// SIMATIC S7-200 SMART project (STEP 7-Micro/WIN SMART), CPU ST40

SYMBOL_TABLE Table 1
Move_X           Q0.0
Move_Z           Q0.1
Grab             Q0.2
Lids_conveyor    Q0.3
Clamp_lid        Q0.4
Pos_raise_lids   Q0.5
Bases_conveyor   Q0.6
Clamp_base       Q0.7
Pos_raise_bases  Q1.0
Strat_light      Q1.1
Reset_light      Q1.2
Stop_light       Q1.3
Counter          QW4
Moving_X         V0.0
Lid_at_place     V0.1
Item_detected    V0.2
Moving_Z         V0.3
Lid_clamped      V0.4
Pos_at_limit_lids V0.5
Base_at_place    V0.6
Base_clamped     V0.7
Pos_at_limit_bases V1.0
Part_leaving     V1.1
Start            V1.2
Reset            V1.3
Stop_            V1.4
Emergency_stop   V1.5
END_SYMBOL_TABLE

SYMBOL_TABLE System Symbols
Always_On        SM0.0    // Always ON
END_SYMBOL_TABLE

ORGANIZATION_BLOCK MAIN:OB1
TITLE=Program Comments
BEGIN
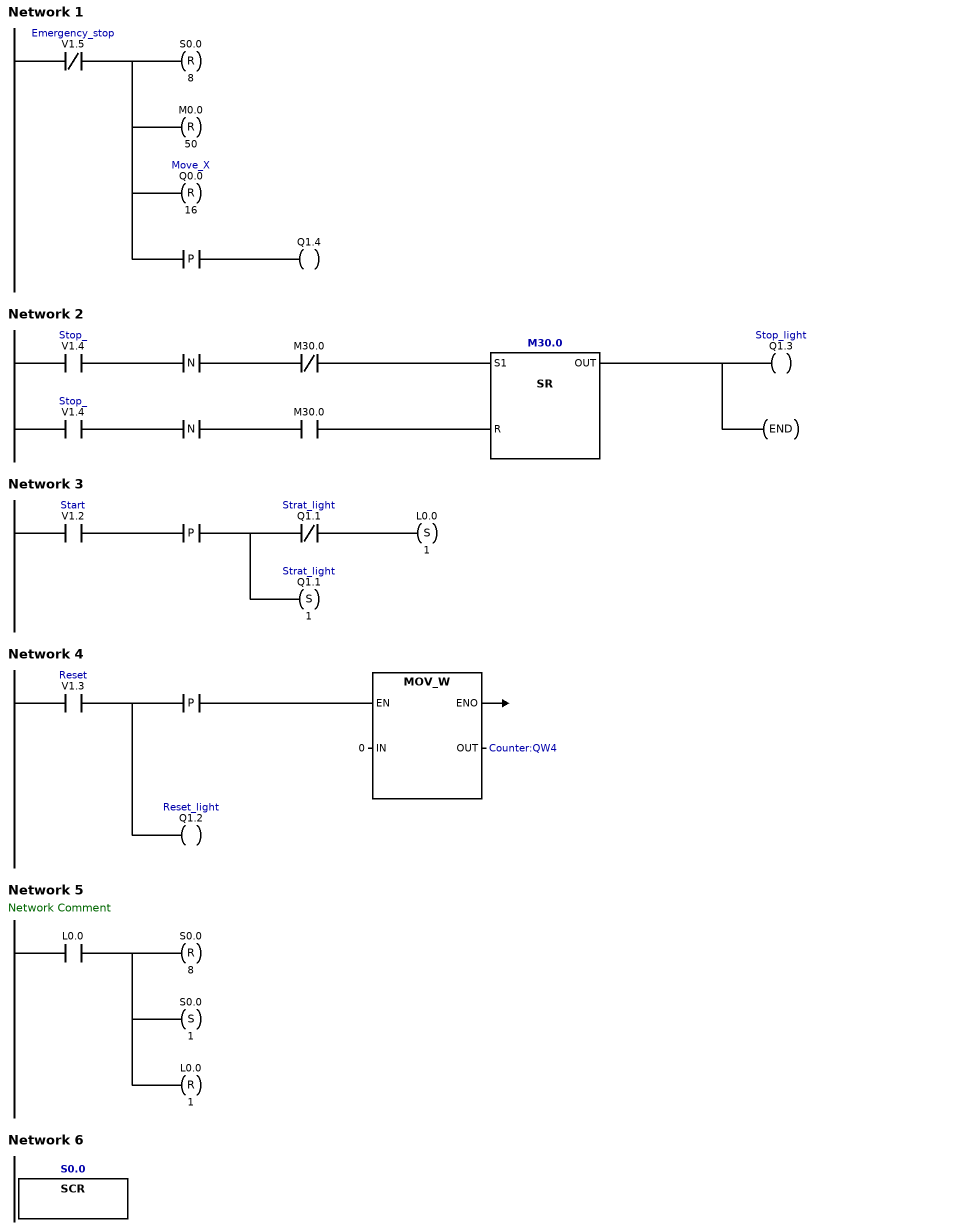
Network 1
LDN    Emergency_stop:V1.5
R      S0.0, 8
R      M0.0, 50
R      Move_X:Q0.0, 16
EU
=      Q1.4
Network 2
LD     Stop_:V1.4
ED
AN     M30.0
LD     Stop_:V1.4
ED
A      M30.0
NOT
A      M30.0
OLD
=      M30.0
=      Stop_light:Q1.3
END
Network 3
LD     Start:V1.2
EU
LPS
AN     Strat_light:Q1.1
S      L0.0, 1
LPP
S      Strat_light:Q1.1, 1
Network 4
LD     Reset:V1.3
LPS
EU
MOVW   0, Counter:QW4
LPP
=      Reset_light:Q1.2
Network 5
// Network Comment
LD     L0.0
R      S0.0, 8
S      S0.0, 1
R      L0.0, 1
Network 6
LSCR   S0.0
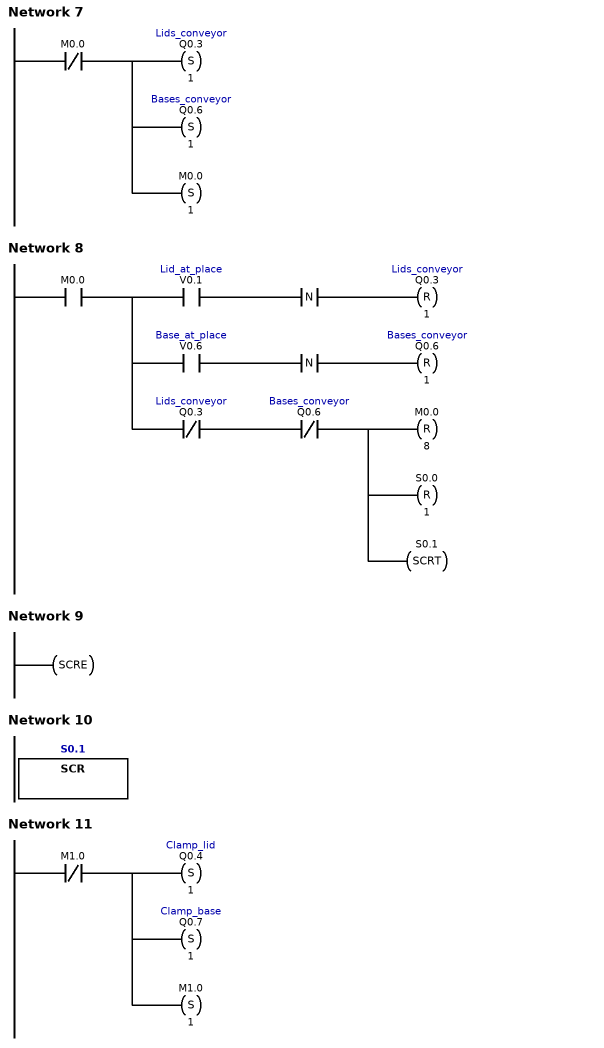
Network 7
LDN    M0.0
S      Lids_conveyor:Q0.3, 1
S      Bases_conveyor:Q0.6, 1
S      M0.0, 1
Network 8
LD     M0.0
LPS
A      Lid_at_place:V0.1
ED
R      Lids_conveyor:Q0.3, 1
LRD
A      Base_at_place:V0.6
ED
R      Bases_conveyor:Q0.6, 1
LPP
AN     Lids_conveyor:Q0.3
AN     Bases_conveyor:Q0.6
R      M0.0, 8
R      S0.0, 1
SCRT   S0.1
Network 9
SCRE
Network 10
LSCR   S0.1
Network 11
LDN    M1.0
S      Clamp_lid:Q0.4, 1
S      Clamp_base:Q0.7, 1
S      M1.0, 1
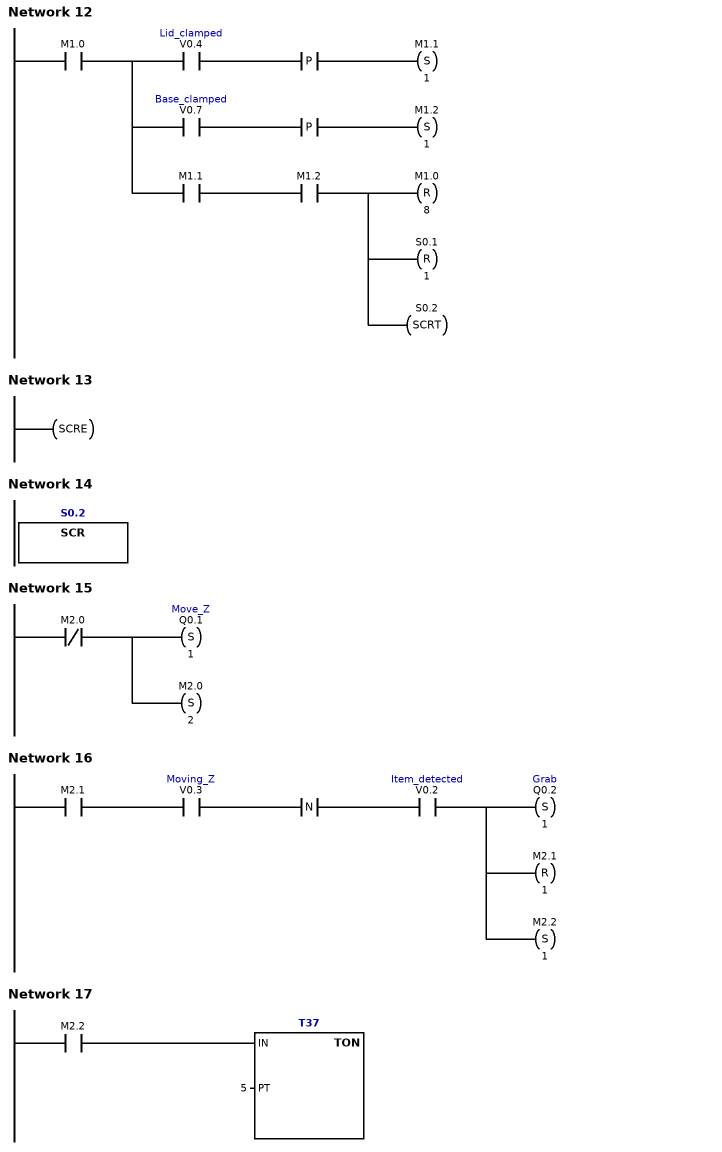
Network 12
LD     M1.0
LPS
A      Lid_clamped:V0.4
EU
S      M1.1, 1
LRD
A      Base_clamped:V0.7
EU
S      M1.2, 1
LPP
A      M1.1
A      M1.2
R      M1.0, 8
R      S0.1, 1
SCRT   S0.2
Network 13
SCRE
Network 14
LSCR   S0.2
Network 15
LDN    M2.0
S      Move_Z:Q0.1, 1
S      M2.0, 2
Network 16
LD     M2.1
A      Moving_Z:V0.3
ED
A      Item_detected:V0.2
S      Grab:Q0.2, 1
R      M2.1, 1
S      M2.2, 1
Network 17
LD     M2.2
TON    T37, 5
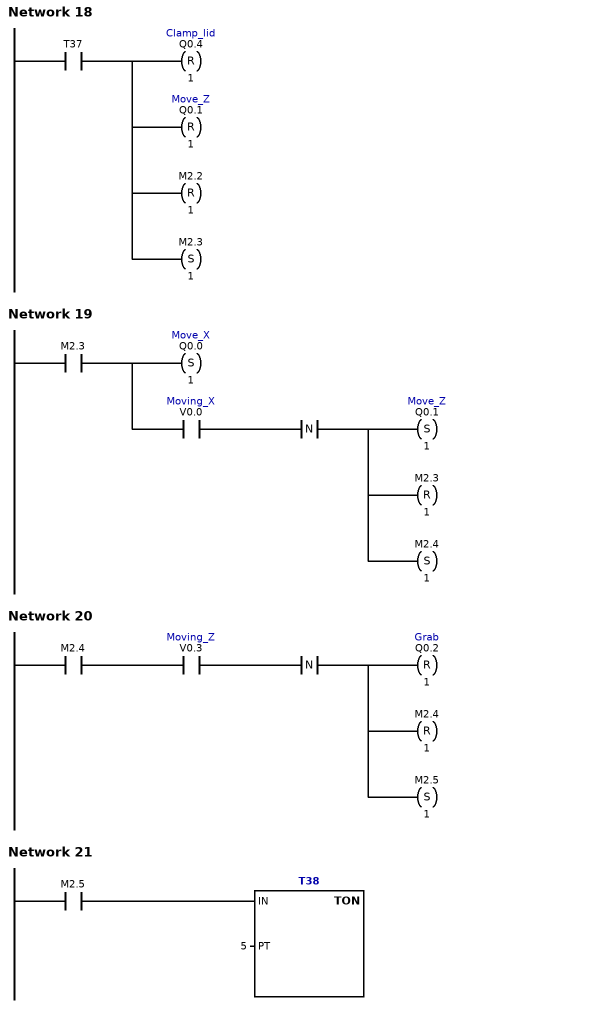
Network 18
LD     T37
R      Clamp_lid:Q0.4, 1
R      Move_Z:Q0.1, 1
R      M2.2, 1
S      M2.3, 1
Network 19
LD     M2.3
S      Move_X:Q0.0, 1
A      Moving_X:V0.0
ED
S      Move_Z:Q0.1, 1
R      M2.3, 1
S      M2.4, 1
Network 20
LD     M2.4
A      Moving_Z:V0.3
ED
R      Grab:Q0.2, 1
R      M2.4, 1
S      M2.5, 1
Network 21
LD     M2.5
TON    T38, 5
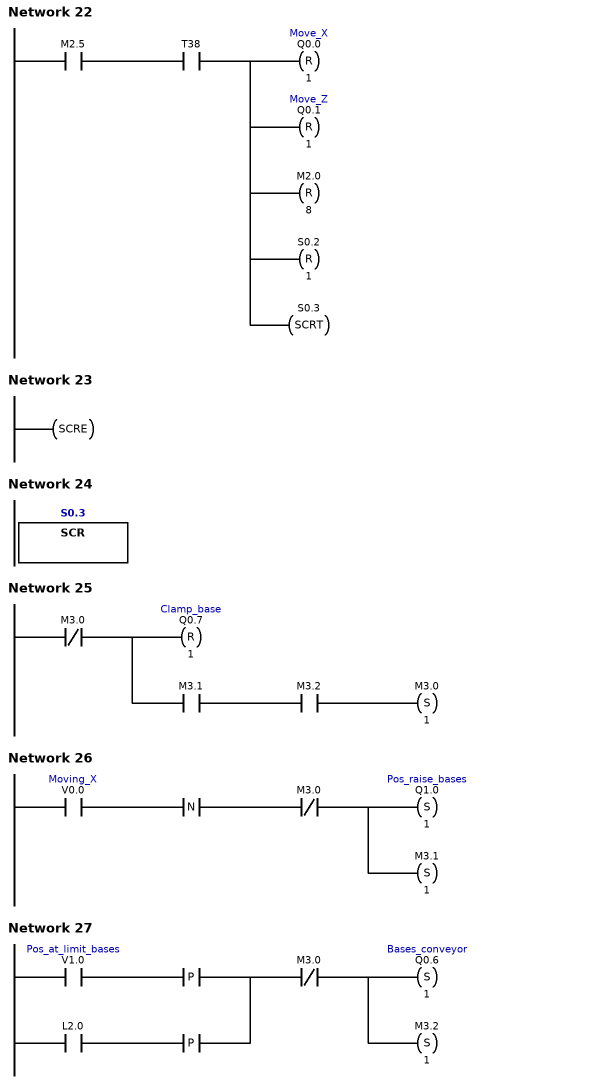
Network 22
LD     M2.5
A      T38
R      Move_X:Q0.0, 1
R      Move_Z:Q0.1, 1
R      M2.0, 8
R      S0.2, 1
SCRT   S0.3
Network 23
SCRE
Network 24
LSCR   S0.3
Network 25
LDN    M3.0
R      Clamp_base:Q0.7, 1
A      M3.1
A      M3.2
S      M3.0, 1
Network 26
LD     Moving_X:V0.0
ED
AN     M3.0
S      Pos_raise_bases:Q1.0, 1
S      M3.1, 1
Network 27
LD     Pos_at_limit_bases:V1.0
EU
LD     L2.0
EU
OLD
AN     M3.0
S      Bases_conveyor:Q0.6, 1
S      M3.2, 1
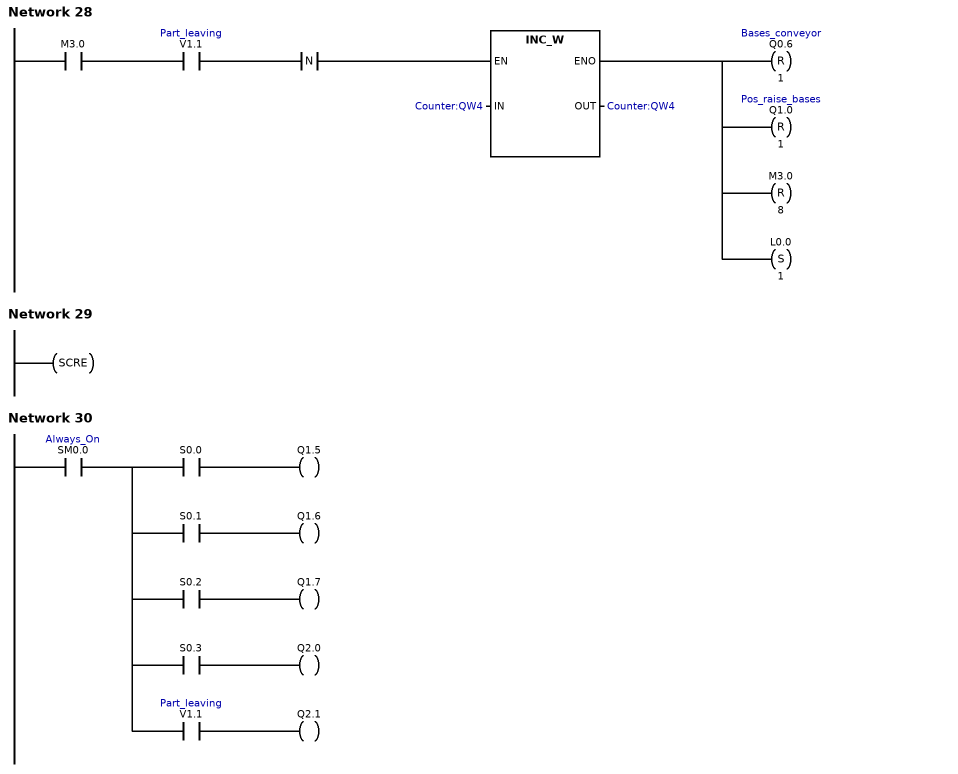
Network 28
LD     M3.0
A      Part_leaving:V1.1
ED
INCW   Counter:QW4
AENO
R      Bases_conveyor:Q0.6, 1
R      Pos_raise_bases:Q1.0, 1
R      M3.0, 8
S      L0.0, 1
Network 29
SCRE
Network 30
LD     Always_On:SM0.0
LPS
A      S0.0
=      Q1.5
LRD
A      S0.1
=      Q1.6
LRD
A      S0.2
=      Q1.7
LRD
A      S0.3
=      Q2.0
LPP
A      Part_leaving:V1.1
=      Q2.1
END_ORGANIZATION_BLOCK
